PROGRAM Axis04_Manual
VAR
//System_Bit
	Always_ON	:	BOOL	:=TRUE	;//상시 ON 
	Always_OFF	:	BOOL	:=FALSE	;//상시 OFF

END_VAR
VAR // added by the converter: edge detectors and wires of the graphical bodies
    _rt1, _rt2 : R_TRIG;
END_VAR

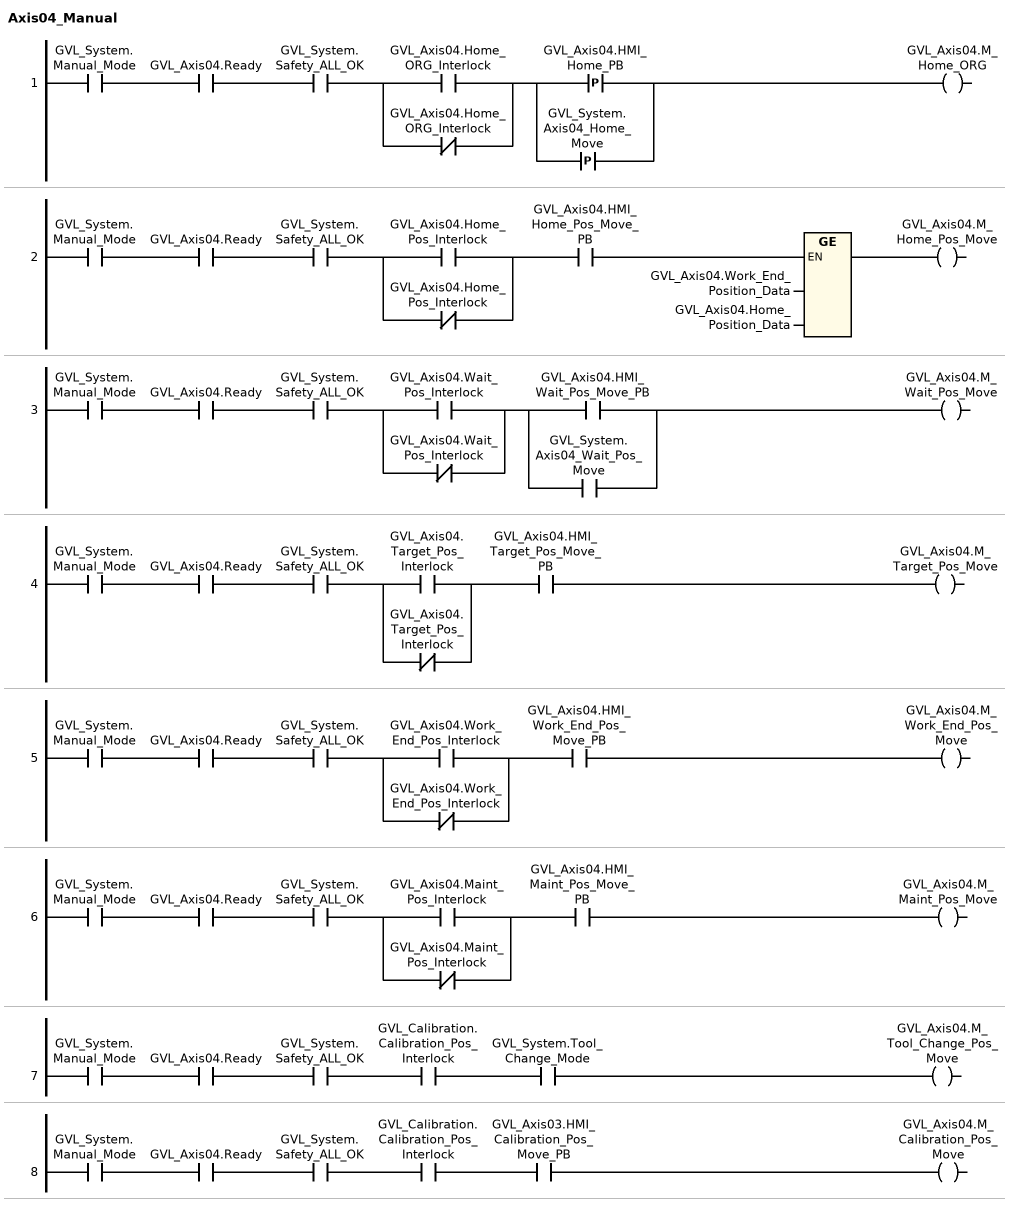
// NETWORK 1
_rt1(CLK := GVL_Axis04.HMI_Home_PB);
_rt2(CLK := GVL_System.Axis04_Home_Move);
GVL_Axis04.M_Home_ORG := GVL_System.Manual_Mode AND GVL_Axis04.Ready AND GVL_System.Safety_ALL_OK AND (GVL_Axis04.Home_ORG_Interlock OR NOT GVL_Axis04.Home_ORG_Interlock) AND (_rt1.Q OR _rt2.Q);

// NETWORK 2
GVL_Axis04.M_Home_Pos_Move := GVL_System.Manual_Mode AND GVL_Axis04.Ready AND GVL_System.Safety_ALL_OK AND (GVL_Axis04.Home_Pos_Interlock OR NOT GVL_Axis04.Home_Pos_Interlock) AND GVL_Axis04.HMI_Home_Pos_Move_PB AND GVL_Axis04.Work_End_Position_Data >= GVL_Axis04.Home_Position_Data;

// NETWORK 3
GVL_Axis04.M_Wait_Pos_Move := GVL_System.Manual_Mode AND GVL_Axis04.Ready AND GVL_System.Safety_ALL_OK AND (GVL_Axis04.Wait_Pos_Interlock OR NOT GVL_Axis04.Wait_Pos_Interlock) AND (GVL_Axis04.HMI_Wait_Pos_Move_PB OR GVL_System.Axis04_Wait_Pos_Move);

// NETWORK 4
GVL_Axis04.M_Target_Pos_Move := GVL_System.Manual_Mode AND GVL_Axis04.Ready AND GVL_System.Safety_ALL_OK AND (GVL_Axis04.Target_Pos_Interlock OR NOT GVL_Axis04.Target_Pos_Interlock) AND GVL_Axis04.HMI_Target_Pos_Move_PB;

// NETWORK 5
GVL_Axis04.M_Work_End_Pos_Move := GVL_System.Manual_Mode AND GVL_Axis04.Ready AND GVL_System.Safety_ALL_OK AND (GVL_Axis04.Work_End_Pos_Interlock OR NOT GVL_Axis04.Work_End_Pos_Interlock) AND GVL_Axis04.HMI_Work_End_Pos_Move_PB;

// NETWORK 6
GVL_Axis04.M_Maint_Pos_Move := GVL_System.Manual_Mode AND GVL_Axis04.Ready AND GVL_System.Safety_ALL_OK AND (GVL_Axis04.Maint_Pos_Interlock OR NOT GVL_Axis04.Maint_Pos_Interlock) AND GVL_Axis04.HMI_Maint_Pos_Move_PB;

// NETWORK 7
GVL_Axis04.M_Tool_Change_Pos_Move := GVL_System.Manual_Mode AND GVL_Axis04.Ready AND GVL_System.Safety_ALL_OK AND GVL_Calibration.Calibration_Pos_Interlock AND GVL_System.Tool_Change_Mode;

// NETWORK 8
GVL_Axis04.M_Calibration_Pos_Move := GVL_System.Manual_Mode AND GVL_Axis04.Ready AND GVL_System.Safety_ALL_OK AND GVL_Calibration.Calibration_Pos_Interlock AND GVL_Axis03.HMI_Calibration_Pos_Move_PB;

END_PROGRAM

(* stored: Version 1.1.0.1, ProductVersion 3.1.4024.15
   POU Axis04_Manual: Id {0bc47764-b7c2-4f2e-b58d-d775da31f11d}, SpecialFunc None *)
